TYPE ANA_DevStd_Prom :
STRUCT
	Value_Mean				: REAL ;	(* (-) Analogic mean value			*)
	Value_Devstd			: REAL ;	(* (-) Standard deviation value		*)
	
	MesAlarmCode			: WORD ;	(* (NA) Internal Akuo AlarmCode     *)
	MesWarningCode			: WORD ;    (* (NA) Internal Akuo WarningCode   *)
	MesEventCode			: WORD ;    (* (NA) Internal Akuo EventCode		*)

END_STRUCT
END_TYPE

(* stored: Version 1.1.0.1, ProductVersion 3.1.4024.11
   DUT ANA_DevStd_Prom: Id {527d27b4-63b2-47bd-a2ec-fc52f5c90934} *)
